# EPICS substitutions: tc32simApp/Db/TC32-sim.substitutions
# TC-32 simulator substitution file.
# Generates TC32-sim.db from tc32-sim-meta.template and temperature-sim.template.
# Structure matches TC32-alsu.substitutions used in the production TCMD IOC.

global {SCAN=$(SCAN), PREC=$(PREC)}

file "tc32-sim-meta.template"
{
pattern {} {}
}

file "temperature-sim.template"
{
pattern
{    R, ADDR,  LOPR,   HOPR, LOLO,  LOW,  HIGH,  HIHI}
{  Ti0,   00,  -270,   1372,    0,   10,    45,    60}
{  Ti1,   01,  -270,   1372,    0,   10,    45,    60}
{  Ti2,   02,  -270,   1372,    0,   10,    45,    60}
{  Ti3,   03,  -270,   1372,    0,   10,    45,    60}
{  Ti4,   04,  -270,   1372,    0,   10,    45,    60}
{  Ti5,   05,  -270,   1372,    0,   10,    45,    60}
{  Ti6,   06,  -270,   1372,    0,   10,    45,    60}
{  Ti7,   07,  -270,   1372,    0,   10,    45,    60}
{  Ti8,   08,  -270,   1372,    0,   10,    45,    60}
{  Ti9,   09,  -270,   1372,    0,   10,    45,    60}
{ Ti10,   10,  -270,   1372,    0,   10,    45,    60}
{ Ti11,   11,  -270,   1372,    0,   10,    45,    60}
{ Ti12,   12,  -270,   1372,    0,   10,    45,    60}
{ Ti13,   13,  -270,   1372,    0,   10,    45,    60}
{ Ti14,   14,  -270,   1372,    0,   10,    45,    60}
{ Ti15,   15,  -270,   1372,    0,   10,    45,    60}
{ Ti16,   16,  -270,   1372,    0,   10,    45,    60}
{ Ti17,   17,  -270,   1372,    0,   10,    45,    60}
{ Ti18,   18,  -270,   1372,    0,   10,    45,    60}
{ Ti19,   19,  -270,   1372,    0,   10,    45,    60}
{ Ti20,   20,  -270,   1372,    0,   10,    45,    60}
{ Ti21,   21,  -270,   1372,    0,   10,    45,    60}
{ Ti22,   22,  -270,   1372,    0,   10,    45,    60}
{ Ti23,   23,  -270,   1372,    0,   10,    45,    60}
{ Ti24,   24,  -270,   1372,    0,   10,    45,    60}
{ Ti25,   25,  -270,   1372,    0,   10,    45,    60}
{ Ti26,   26,  -270,   1372,    0,   10,    45,    60}
{ Ti27,   27,  -270,   1372,    0,   10,    45,    60}
{ Ti28,   28,  -270,   1372,    0,   10,    45,    60}
{ Ti29,   29,  -270,   1372,    0,   10,    45,    60}
{ Ti30,   30,  -270,   1372,    0,   10,    45,    60}
{ Ti31,   31,  -270,   1372,    0,   10,    45,    60}
}
